// TIA Portal V18 export
FUNCTION "TEMPLATE--v1.1--02_EM Push Button" : Void   // FC5, F_LAD
TITLE = Mirror PB
{ S7_Optimized_Access := 'TRUE' }
// v1.0 First emission
// 1.1 Aligned Syntax to signal_types.csv of the py_builder
BEGIN

REGION Network 1: !!NetworkComment$$
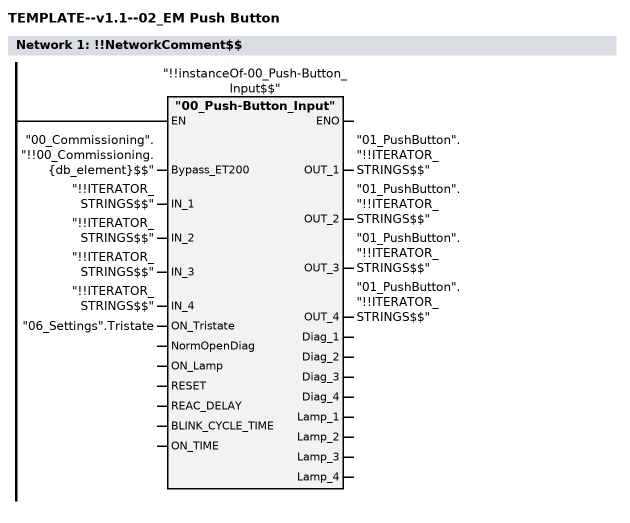
   RUNG wire#powerrail
      "!!instanceOf-00_Push-Button_Input$$"(Bypass_ET200 := "00_Commissioning"."!!00_Commissioning.{db_element}$$", IN_1 := "!!ITERATOR_STRINGS$$", IN_2 := "!!ITERATOR_STRINGS$$", IN_3 := "!!ITERATOR_STRINGS$$", IN_4 := "!!ITERATOR_STRINGS$$", ON_Tristate := "06_Settings".Tristate, NormOpenDiag :=, ON_Lamp :=, RESET :=, REAC_DELAY :=, BLINK_CYCLE_TIME :=, ON_TIME :=, OUT_1 => "01_PushButton"."!!ITERATOR_STRINGS$$", OUT_2 => "01_PushButton"."!!ITERATOR_STRINGS$$", OUT_3 => "01_PushButton"."!!ITERATOR_STRINGS$$", OUT_4 => "01_PushButton"."!!ITERATOR_STRINGS$$", Diag_1 =>, Diag_2 =>, Diag_3 =>, Diag_4 =>, Lamp_1 =>, Lamp_2 =>, Lamp_3 =>, Lamp_4 =>)
   END_RUNG
   // the same network as SCL:
   "!!instanceOf-00_Push-Button_Input$$"(Bypass_ET200 := "00_Commissioning"."!!00_Commissioning.{db_element}$$",   // "00_Push-Button_Input"
                           IN_1 := "!!ITERATOR_STRINGS$$",
                           IN_2 := "!!ITERATOR_STRINGS$$",
                           IN_3 := "!!ITERATOR_STRINGS$$",
                           IN_4 := "!!ITERATOR_STRINGS$$",
                           ON_Tristate := "06_Settings".Tristate,
                           OUT_1 => "01_PushButton"."!!ITERATOR_STRINGS$$",
                           OUT_2 => "01_PushButton"."!!ITERATOR_STRINGS$$",
                           OUT_3 => "01_PushButton"."!!ITERATOR_STRINGS$$",
                           OUT_4 => "01_PushButton"."!!ITERATOR_STRINGS$$");
END_REGION
END_FUNCTION
